TYPE T_DiskLoggerPath : STRING(PARAM_Constants.DISK_LOGGER_PATH_LENGTH); END_TYPE

(* stored: Version 1.1.0.1
   DUT T_DiskLoggerPath: Id {4374c226-db05-0521-3feb-7cbb42f6de32} *)
